FUNCTION_BLOCK fbXYMoverEM EXTENDS fbEM

// TEST
em.Config.Data.Q[6] := true;

END_FUNCTION_BLOCK

(* stored: Version 1.1.0.1, ProductVersion 3.1.4024.12
   POU fbXYMoverEM: Id {542faac4-2fc2-4de1-969d-21d2b14af459}, SpecialFunc None *)
